// TIA Portal V16 export
// export: Created 2021-05-12T14:39:33.3108571Z, ExportSetting WithDefaults, DisplayName Totally Integrated Automation Portal, DisplayVersion V16 Update 3, DisplayName TIA Portal Version Control Interface, DisplayVersion V16 Update 2, DisplayName TIA Portal Openness, DisplayVersion V16 Update 3, DisplayName STEP 7 Professional, DisplayVersion V16 Update 3, DisplayName STEP 7 Safety, DisplayVersion V16, DisplayName WinCC Professional, DisplayVersion V16 Update 3
DATA_BLOCK "DB21001_Dy_SysGlobalData"   // DB21001
TITLE = Dynamic DB — Sys - Global Data
{ S7_Optimized_Access := 'TRUE' }
AUTHOR : M_Gledhill
FAMILY : System
NAME : Dy_SysGlobalData
VERSION : 1.0
// PRACTICAL SERIES AUTOMATION LIBRARY (PAL)   —   COPYRIGHT 2020 – M. GLEDHILL (MIT LICENCE)
//                   ———— ◆ ————
//  FOR DETAILED DOCUMENTATION — SELECT THE BLOCK IN THE PROJECT TREE AND PRESS SHIFT + F1
//  FULL ONLINE DOCUMENTATION IS AVAILABLE AT: https://practicalseries.com/2001-pal/index.html
// stored: AutoNumber false, DBAccessibleFromOPCUA true, IsOnlyStoredInLoadMemory false, IsRetainMemResEnabled false, IsWriteProtectedInAS false, MemoryReserve 100
   VAR
      _DB_Header { ExternalWritable := 'False'} : Array[0..79] of Bool;   // STANDARD SYSTEM GLOBAL DATA
      __________0000_0 { ExternalWritable := 'False'} : Bool := false;
      __________0000_1 { ExternalWritable := 'False'} : Bool := false;   // ▀▀▀▀ DB CURRENT REVISION
      revInfo { ExternalWritable := 'False'} : "UT01000_St_SysRevision";
      __________0010_0 { ExternalWritable := 'False'} : Bool := false;
      __________0010_1 { ExternalWritable := 'False'} : Bool := false;   // ▀▀▀▀ PROJECT CURRENT REVISION
      projRevInfo { ExternalWritable := 'False'} : "UT01000_St_SysRevision";
      __________0020_0 { ExternalWritable := 'False'} : Bool := false;
      __________0020_1 { ExternalWritable := 'False'} : Bool := false;   // ▀▀▀▀ SYSTEM SIGNALS — LOGIC AND TIMING SIGNALS
      SysSignals { ExternalWritable := 'False'} : "UT21000_Dy_SysSignals";
      __________0030_0 { ExternalWritable := 'False'} : Bool := false;
      __________0030_1 { ExternalWritable := 'False'} : Bool := false;   // ▀▀▀▀ SYSTEM DATA — CYCLE TIMING AND RTC
      SysData { ExternalWritable := 'False'} : "UT21001_Dy_SysData";
      __________0040_0 { ExternalWritable := 'False'} : Bool := false;
      __________0040_1 { ExternalWritable := 'False'} : Bool := false;   // ▀▀▀▀ OB CALL TIMES
      OB10_CallTime { ExternalWritable := 'False'} : DTL;   // Time of day interrupt 1
      OB11_CallTime { ExternalWritable := 'False'} : DTL;   // Time of day interrupt 2
      OB12_CallTime { ExternalWritable := 'False'} : DTL;   // Time of day interrupt 3
      OB13_CallTime { ExternalWritable := 'False'} : DTL;   // Time of day interrupt 4
      OB14_CallTime { ExternalWritable := 'False'} : DTL;   // Time of day interrupt 5
      OB15_CallTime { ExternalWritable := 'False'} : DTL;   // Time of day interrupt 6
      OB16_CallTime { ExternalWritable := 'False'} : DTL;   // Time of day interrupt 7
      OB17_CallTime { ExternalWritable := 'False'} : DTL;   // Time of day interrupt 8
      OB20_CallTime { ExternalWritable := 'False'} : DTL;   // Time delay interrupt 1
      OB21_CallTime { ExternalWritable := 'False'} : DTL;   // Time delay interrupt 2
      OB22_CallTime { ExternalWritable := 'False'} : DTL;   // Time delay interrupt 3
      OB23_CallTime { ExternalWritable := 'False'} : DTL;   // Time delay interrupt 4
      OB30_CallTime { ExternalWritable := 'False'} : DTL;   // Timed cyclic interrupt 1
      OB31_CallTime { ExternalWritable := 'False'} : DTL;   // Timed cyclic interrupt 2
      OB32_CallTime { ExternalWritable := 'False'} : DTL;   // Timed cyclic interrupt 3
      OB33_CallTime { ExternalWritable := 'False'} : DTL;   // Timed cyclic interrupt 4
      OB34_CallTime { ExternalWritable := 'False'} : DTL;   // Timed cyclic interrupt 5
      OB35_CallTime { ExternalWritable := 'False'} : DTL;   // Timed cyclic interrupt 6
      OB36_CallTime { ExternalWritable := 'False'} : DTL;   // Timed cyclic interrupt 7
      OB37_CallTime { ExternalWritable := 'False'} : DTL;   // Timed cyclic interrupt 8
      OB38_CallTime { ExternalWritable := 'False'} : DTL;   // Timed cyclic interrupt 9
      OB40_CallTime { ExternalWritable := 'False'} : DTL;   // Hardware interrupt 1
      OB41_CallTime { ExternalWritable := 'False'} : DTL;   // Hardware interrupt 2
      OB42_CallTime { ExternalWritable := 'False'} : DTL;   // Hardware interrupt 3
      OB43_CallTime { ExternalWritable := 'False'} : DTL;   // Hardware interrupt 4
      OB44_CallTime { ExternalWritable := 'False'} : DTL;   // Hardware interrupt 5
      OB45_CallTime { ExternalWritable := 'False'} : DTL;   // Hardware interrupt 6
      OB46_CallTime { ExternalWritable := 'False'} : DTL;   // Hardware interrupt 7
      OB47_CallTime { ExternalWritable := 'False'} : DTL;   // Hardware interrupt 8
      OB80_CallTime { ExternalWritable := 'False'} : DTL;   // Error interrupt — max cycle time exceeded
      OB82_CallTime { ExternalWritable := 'False'} : DTL;   // Error interrupt — module diagnostic
      OB83_CallTime { ExternalWritable := 'False'} : DTL;   // Error interrupt — module changed
      OB86_CallTime { ExternalWritable := 'False'} : DTL;   // Error interrupt — rack fault
      OB100_CallTime { ExternalWritable := 'False'} : DTL;   // Start-up interrupt
      OB121_CallTime { ExternalWritable := 'False'} : DTL;   // Error interrupt — programming fault
      OB122_CallTime { ExternalWritable := 'False'} : DTL;   // Error interrupt — IO access fault
   END_VAR
BEGIN
   // _DB_Header[0] : ▀▀▀▀▀▀▀▀▀▀▀▀▀▀▀▀▀▀▀▀▀▀▀▀▀▀▀▀▀▀▀▀▀▀▀▀▀▀▀▀▀▀▀▀
   // _DB_Header[2] : TITLE: STANDARD SYSTEM GLOBAL DATA
   // _DB_Header[4] : ▄▄▄▄▄▄▄▄▄▄▄▄▄▄▄▄▄▄▄▄▄▄▄▄▄▄▄▄▄▄▄▄▄▄▄▄▄▄▄▄▄▄▄▄
   // _DB_Header[5] : TYPE: DYNAMIC
   // _DB_Header[6] : ▀▀▀▀▀▀▀▀▀▀▀▀▀▀▀▀▀▀▀▀▀▀▀▀▀▀▀▀▀▀▀▀▀▀▀▀▀▀▀▀▀▀▀▀
   // _DB_Header[8] : Global system data storage DB. The block records various system variables and information:
   // _DB_Header[10] : • Project revision data
   // _DB_Header[11] : • Common system signals (logic and timing)
   // _DB_Header[12] : • Cycle timing information (previous, max, min and a cycle counter)
   // _DB_Header[13] : • CPU real time clock data (in globally readable format)
   // _DB_Header[14] : • Last call time of any interrupt OB
   // _DB_Header[16] : The cycle timing information and the RTC data are provided by FC01000. The interrupt OB data
   // _DB_Header[17] : is provided by the individual OBs.
   // _DB_Header[19] : ━━━ ⬙⬙⬙⬙⬙⬙ ━━━
   // _DB_Header[21] : ▄▄▄▄▄▄▄▄▄▄▄▄▄▄▄▄▄▄▄▄▄▄▄▄▄▄▄▄▄▄▄▄▄▄▄▄▄▄▄▄▄▄▄▄
   // _DB_Header[22] : MODIFICATION HISTORY
   // _DB_Header[24] : This is a summary of the recent software modifications made to this block (most recent at top)
   // _DB_Header[26] : ―――――――――――――――――――――――――――――――――――――――――――
   // _DB_Header[27] : DATE REVISION MASTER BRANCH DEV
   // _DB_Header[28] : (nnn.amm) COMMIT TAG (Base ---> Merge) BRANCH Author
   // _DB_Header[29] : ———————————————————————————————————————————
   // _DB_Header[30] : 2021.05.11 001.000 D0006 D0005 D0006 None M. Gledhill
   // _DB_Header[31] : FC01001 — RELEASED FOR USE
   // _DB_Header[32] : Merge back to master branch
   // _DB_Header[34] : 2021.05.11 000.801 D0005A-000.801 D0005 N/A D0005A M. Gledhill
   // _DB_Header[35] : FC01001 — Released for SMT
   // _DB_Header[37] : 2021.05.08 000.101 D0005A-000.101 D0005 N/A D0005A M. Gledhill
   // _DB_Header[38] : FC01001 Migration to VCS
   // _DB_Header[39] : ———————————————————————————————————————————
   // _DB_Header[41] : ██████████████ █ █ █ █ END █ █ █ █ ██████████████
   revInfo.REV_BLOCK := 'DB21001';
   revInfo.REV_NUMBER := '001.000';
   revInfo.REV_DATE := '2021-05-11';
   revInfo.REV_AUTHOR := 'M. Gledhill';
END_DATA_BLOCK
